FUNCTION_BLOCK FB_CheckPistonPosition
VAR_INPUT
END_VAR
VAR_OUTPUT
END_VAR
VAR
END_VAR

// Check if piston is out of bounds
IF HMI.fCylinderPositon > Parameters.stPistonRange.fPistonPosMax THEN
	HMI.fCylinderPositon := Parameters.stPistonRange.fPistonPosMax;	
	HMI.sPistonEndStopMessage := Parameters.stPistonOutOfBounds.sPistonMax;
	Parameters.eErrorModes := E_ErrorModes.MaxLimit;
	HMI.sPistonEndStopMessage := Parameters.stPistonOutOfBounds.sPistonMax;
ELSIF HMI.fCylinderPositon < Parameters.stPistonRange.fPistonPosMin  THEN
	HMI.fCylinderPositon := Parameters.stPistonRange.fPistonPosMin;
	Parameters.eErrorModes := E_ErrorModes.MinLimit;
	HMI.sPistonEndStopMessage := Parameters.stPistonOutOfBounds.sPistonMin;
ELSE
	HMI.sPistonEndStopMessage := Parameters.stPistonOutOfBounds.sNotActive;
	Parameters.eErrorModes := E_ErrorModes.NaN;
END_IF

END_FUNCTION_BLOCK

(* stored: Version 1.1.0.1, ProductVersion 3.1.4024.10
   POU FB_CheckPistonPosition: Id {e27b36ef-4a24-48d6-828c-722716f11070}, SpecialFunc None *)
